ORGANIZATION_BLOCK 主程序:OB1
TITLE=程序注释
BEGIN
Network 1 // 网络标题
// 主程序
LD     SM0.1
CALL   SBR0
Network 2
// 子程序
LD     SM0.1
MOVB   16#F8, SMB47
HDEF   1, 11
MOVD   +0, SMD48
MOVD   +50, SMD52
ATCH   INT0, 13
ENI
HSC    1
END_ORGANIZATION_BLOCK
SUBROUTINE_BLOCK SBR_0:SBR0
TITLE=子程序注释
BEGIN
Network 1 // 网络标题
// 网络注释
END_SUBROUTINE_BLOCK
INTERRUPT_BLOCK INT_0:INT0
TITLE=中断程序注释
BEGIN
Network 1 // 网络标题
// 网络注释
END_INTERRUPT_BLOCK
